// SIMATIC STEP 7 (V5.x) project YieldCalculation
// CPU: CPU414-2 DP(1)
// station: P_ADR_BUS
// station: 硬件
// station: SIMATIC 400 站点
// program: S7 程序(1)

SYMBOL_TABLE
"Cycle Execution"	OB 1	OB 1
"READ_CLK"	SFC 1	SFC 1	// Read System Clock
END_SYMBOL_TABLE

FUNCTION_BLOCK FB 2800
TITLE = YieldCalculation
//
//主要用于计算班、年、月、日产量， 
//增加早班、中班、晚班每两小时的产量计算
//
AUTHOR : QIAO
FAMILY : QFam
NAME : ProCount
VERSION : 1.3
VAR_INPUT
  Product_Total : REAL ;
  Initialize : BOOL ;
END_VAR
VAR_OUTPUT
  Product_Early_Class : REAL ;	//早班产量（9:00-17:00）
  Product_Middle_Class : REAL ;	//中班产量（17:00-1:00）
  Product_Late_Class : REAL ;	//晚班产量（1:00-9:00）
  Product_Day : REAL ;	//日产量
  Product_Month : REAL ;	//月产量
  Product_Year : REAL ;	//年产量
  Product_LastMonth : REAL ;	//上月产量
  Product_Yesterday : REAL ;	//昨天产量
  Product_Early_2H_1 : REAL ;	//早班第一段(9:00-11:00)
  Product_Early_2H_2 : REAL ;	//早班第二段(11:00-13:00)
  Product_Early_2H_3 : REAL ;	//早班第三段(13:00-15:00)
  Product_Early_2H_4 : REAL ;	//早班第四段(15:00-17:00)
  Product_Middle_2H_1 : REAL ;	//中班第一段(17:00-19:00)
  Product_Middle_2H_2 : REAL ;	//中班第二段(19:00-21:00)
  Product_Middle_2H_3 : REAL ;	//中班第三段(21:00-23:00)
  Product_Middle_2H_4 : REAL ;	//中班第四段(23:00-1:00)
  Product_Late_2H_1 : REAL ;	//晚班第一段(1:00-3:00)
  Product_Late_2H_2 : REAL ;	//晚班班第二段(3:00-5:00)
  Product_Late_2H_3 : REAL ;	//晚班第三段(5:00-7:00)
  Product_Late_2H_4 : REAL ;	//晚班第四段(7:00-9:00)
  Init_Done : BOOL ;
END_VAR
VAR
  DateAndTimeNow : DATE_AND_TIME ;
  YearNow : INT ;
  MonthNow : INT ;
  DayNow : INT ;
  HourNow : INT ;
  MinuteNow : INT ;
  SecondNow : INT ;
  HourLast : INT ;
  MinuteLast : INT ;
  SecondLast : INT ;
  DayLast : INT ;
  MonthLast : INT ;
  YearLast : INT ;
  MonthNowFormer : INT ;
  YearNowFormer : INT ;
  DayNowFormer : INT ;
  StartEarlyClassPro : REAL ;
  StartMiddleClassPro : REAL ;
  StartLateClassPro : REAL ;
  StartDayClassPro : REAL ;
  StartMonthClassPro : REAL ;
  StartYearClassPro : REAL ;
  StartEarly_2H_1 : REAL ;	//早班第一段(9:00-11:00)
  StartEarly_2H_2 : REAL ;	//早班第二段(11:00-13:00)
  StartEarly_2H_3 : REAL ;	//早班第三段(13:00-15:00)
  StartEarly_2H_4 : REAL ;	//早班第四段(15:00-17:00)
  StartMiddle_2H_1 : REAL ;	//中班第一段(17:00-19:00)
  StartMiddle_2H_2 : REAL ;	//中班第二段(19:00-21:00)
  StartMiddle_2H_3 : REAL ;	//中班第三段(21:00-23:00)
  StartMiddle_2H_4 : REAL ;	//中班第四段(23:00-1:00)
  StartLate_2H_1 : REAL ;	//晚班第一段(1:00-3:00)
  StartLate_2H_2 : REAL ;	//晚班第二段(3:00-5:00)
  StartLate_2H_3 : REAL ;	//晚班第三段(5:00-7:00)
  StartLate_2H_4 : REAL ;	//晚班第四段(7:00-9:00)
  Early_2H_1_Flag : BOOL ;
  Early_2H_2_Flag : BOOL ;
  Early_2H_3_Flag : BOOL ;
  Early_2H_4_Flag : BOOL ;
  Middle_2H_1_Flag : BOOL ;
  Middle_2H_2_Flag : BOOL ;
  Middle_2H_3_Flag : BOOL ;
  Middle_2H_4_Flag : BOOL ;
  Late_2H_1_Flag : BOOL ;
  Late_2H_2_Flag : BOOL ;
  Late_2H_3_Flag : BOOL ;
  Late_2H_4_Flag : BOOL ;
  IsFirstScan : BOOL  := TRUE;
  EarlyClassFlag : BOOL ;
  MiddleClassFlag : BOOL ;
  LateClassFlag : BOOL ;
  DayFlag : BOOL ;
  MonthFlag : BOOL ;
  YearFlag : BOOL ;
  LastMonth_Total : REAL ;
  Yesterday_Total : REAL ;
END_VAR
VAR_TEMP
  Read_Return : INT ;
END_VAR
BEGIN
// body was compiled from an SCL source; compiled code not shown
END_FUNCTION_BLOCK

FUNCTION_BLOCK FB 2801
TITLE = Test Yield Calculation
//变量声明
VERSION : 0.0
VAR
  Test_Product_Total : REAL ;
  Test_Initialize : BOOL ;
  fbProductCount : FB 2800;
  Test_White_Class : REAL ;
  Test_Night_Class : REAL ;
  Test_Day : REAL ;
  Test_Month : REAL ;
  Test_Year : REAL ;
  Test_Init_Done : BOOL ;
  Test_White_3H_1 : REAL ;
  Test_White_3H_2 : REAL ;
  Test_White_3H_3 : REAL ;
  Test_White_3H_4 : REAL ;
  Test_Night_3H_1 : REAL ;
  Test_Night_3H_2 : REAL ;
  Test_Night_3H_3 : REAL ;
  Test_Night_3H_4 : REAL ;
  Simulate_Time : INT ;
  Test_Step : INT ;
END_VAR
BEGIN
// body was compiled from an SCL source; compiled code not shown
END_FUNCTION_BLOCK

DATA_BLOCK DB 2800
AUTHOR : QIAO
FAMILY : QFam
VERSION : 0.0
FB 2800
BEGIN
END_DATA_BLOCK

DATA_BLOCK DB 2801
VERSION : 0.0
FB 2801
BEGIN
END_DATA_BLOCK

ORGANIZATION_BLOCK "Cycle Execution"	// OB 1
TITLE = "Main Program Sweep (Cycle)"
VERSION : 0.1
VAR_TEMP
  OB1_EV_CLASS : BYTE ;	//Bits 0-3 = 1 (Coming event), Bits 4-7 = 1 (Event class 1)
  OB1_SCAN_1 : BYTE ;	//1 (Cold restart scan 1 of OB 1), 3 (Scan 2-n of OB 1)
  OB1_PRIORITY : BYTE ;	//Priority of OB Execution
  OB1_OB_NUMBR : BYTE ;	//1 (Organization block 1, OB1)
  OB1_RESERVED_1 : BYTE ;	//Reserved for system
  OB1_RESERVED_2 : BYTE ;	//Reserved for system
  OB1_PREV_CYCLE : INT ;	//Cycle time of previous OB1 scan (milliseconds)
  OB1_MIN_CYCLE : INT ;	//Minimum cycle time of OB1 (milliseconds)
  OB1_MAX_CYCLE : INT ;	//Maximum cycle time of OB1 (milliseconds)
  OB1_DATE_TIME : DATE_AND_TIME ;	//Date and time OB1 started
END_VAR
BEGIN
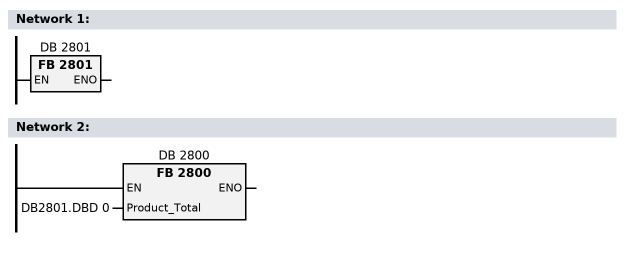
NETWORK
TITLE =
      CALL  FB 2801 , DB 2801;
      NOP   0;
NETWORK
TITLE =
      CALL  FB 2800 , DB 2800 (
           Product_Total            := DB2801.DBD 0);
      NOP   0;
END_ORGANIZATION_BLOCK
